PROGRAM PRG_PROTOTYPE
VAR
END_VAR

//gauges
MR2K3_GPI_1(PG=>);
TV2K4_GPI_1(PG=>);
MR1K4_GPI_1(PG=>);

MR2K3_GCC_1(PG:=MR2K3_GPI_1.PG);
TV2K4_GCC_1(PG:=TV2K4_GPI_1.PG);
MR1K4_GCC_1(PG:=MR1K4_GPI_1.PG);

//valves
TV2K4_VGC_1(i_stUSG := MR2K3_GCC_1.IG, 
			i_stDSG:= TV2K4_GCC_1.IG, 
			i_xDis_DPIlk := TRUE, 
			i_xEPS_OK := TRUE, 
			i_xPMPS_OK := TRUE, 
			i_xExt_OK := TRUE, 
			i_xOverrideMode := xSystemOverrideMode);
			
MR1K4_VGC_1(i_stUSG := TV2K4_GCC_1.IG, 
			i_stDSG:= MR1K4_GCC_1.IG, 
			i_xDis_DPIlk := TRUE, 
			i_xEPS_OK := TRUE, 
			i_xPMPS_OK := TRUE, 
			i_xExt_OK := TRUE, 
			i_xOverrideMode := xSystemOverrideMode);
			
//pumps
TV2KO_PIP_1(i_stGauge:= TV2K4_GCC_1.IG);

END_PROGRAM

(* stored: Version 1.1.0.1, ProductVersion 3.1.4022.12
   POU PRG_PROTOTYPE: Id {eb501625-f746-47fa-ac8c-3ae898c079cf}, SpecialFunc None *)
